FUNCTION linSpdCommandMixer : LREAL
VAR_INPUT
	modeEnable:INT;
    linMoveSpdCommand, linPosErr:LREAL;
END_VAR
VAR
END_VAR

IF(modeEnable=0) THEN
    linSpdCommandMixer:= 0;
	return;
 ELSIF(modeEnable=4  OR modeEnable = 5)THEN
    IF(ABS(linPosErr)<0.005) THEN
       linSpdCommandMixer:=  0;
	   RETURN;
    else
       linSpdCommandMixer:=linMoveSpdCommand;   
	   RETURN;
	END_IF 
  END_IF
  linSpdCommandMixer:=  0;

END_FUNCTION

(* stored: Version 1.1.0.1, ProductVersion 3.1.4024.12
   POU linSpdCommandMixer: Id {b0c81978-755d-467c-93bb-0e8c4fae62fd}, SpecialFunc None *)
